{attribute 'GeneratedUsingTerminal: EK1100-0000-0018'}
{attribute addProperty BoxType "EK1100-0000-0018"}
{attribute addProperty Id "Beckhoff_EP8xxxEK1122Beckhoff_EP8xxxEK1122_58AD3630282"}
{attribute addProperty CRC "3954550627"}
{attribute addProperty Size "282"}
TYPE Beckhoff_EP8xxx_EBB5A763 EXTENDS EK1100_AB5A9467 :
STRUCT
	{attribute addProperty Name "Beckhoff_EP8xxxEK1122"}
	{attribute addProperty PreviousPort "Beckhoff EP8xxx : B"}
	Beckhoff_EP8xxxEK1122 : Beckhoff_EP8xxxEK1122_58AD3630;
END_STRUCT
END_TYPE

(* stored: Version 1.2.0.0, ProductVersion 3.1.4024.9
   DUT Beckhoff_EP8xxx_EBB5A763: Id {211a85d1-6ec3-4930-ab26-ea3ea56c5f41} *)
